KUKA KRL program: chk_w6_grp5_opn.src

&ACCESS RVO6
&COMMENT Check GRP AXOR Z5 OPEN
DEF chk_w6_grp5_opn( )

; Check gripper axor OPEN Z5.1/2/3/4
;//---- Start User-------

$TIMER[10] = 0
$TIMER_STOP[10] = FALSE

WAIT FOR ($IN[501] and $in[503] AND $IN[505] AND $IN[507])
WAIT FOR (NOT $IN[502] and NOT $in[504] AND NOT $IN[506] AND NOT $IN[508])

$TIMER_STOP[10] = TRUE
$TIMER[10] = 0

;//---- End User---------
END
